(* CODESYS project PLCPID.project
   Title: PLCTEST
   Author: Peter
   Version: 0.0.0.21

Project tree, tasks and I/O mapping:
  MyController_1 : TM241CEC24T/U, Schneider Electric, order no. TM241CEC24T/U, version 4.0.6.18
    application Application
      libraries: HMISCU PTOPWM, 2.0.1.4 (Schneider Electric); SM3_Basic, 3.5.3.83 (3S - Smart Software Solutions GmbH)
      task MAST (cyclic, interval 2 ms, priority 15, watchdog 100 ms x 1) calls PIDController
      global variables GVL
      program PIDController [ST]
      function block Home [ST]
    DI : Digital Inputs, Schneider Electric, version 4.0.6.18
        settings: IOs Usage = 3
        input  Application.PIDController.sensor_r : BOOL  // IW0.I6
        input  Application.PIDController.sensor_l : BOOL  // IW0.I7
        input  ibDI_IB1 : BYTE  // IB1
        unmapped channels: IW0
    DQ : Digital Outputs, Schneider Electric, version 4.0.6.18
        output Application.PIDController.en_driver : BOOL  // QW0.Q7
        output Application.PIDController.fault_reset : BOOL  // QW0.Q8
        unmapped channels: QW0, QB1
    Counters : Counters, Schneider Electric, version 4.0.6.18
        settings: Instance name = 'encoder'; B input History = 'old=-1 new=1'; A input History = 'old=-1 new=0'; Temporary Instance name = 'encoder'
    Pulse_Generators : Pulse Generators, Schneider Electric, version 4.0.6.18
        settings: A output History = 'old=7 new=-1'
    Cartridge_1 : Cartridge, Schneider Electric, version 4.0.6.18
    IO_Bus : IO bus - TM3, Schneider Electric, version 4.0.6.18
      Module_1 : TM3SAF5R/G, Schneider Electric, order no. TM3SAF5R/G, version 1.0.1.12
          output Application.PIDController.en_safety : BOOL  // QB0.Enable
          unmapped channels: IW0, QB0
      Module_2 : TM3AQ4/G, Schneider Electric, order no. TM3AQ4/G, version 1.0.0.12
          settings: KPI Configuration.KPI Configuration[0] = 17; KPI Configuration.KPI Configuration[4] = 240; KPI Configuration.KPI Configuration[5] = 216; KPI Configuration.KPI Configuration[12] = 16; KPI Configuration.KPI Configuration[13] = 39
          output Application.PIDController.motor_value : INT  // QW0
          output qiModule_2_QW2 : INT  // QW2
          output qiModule_2_QW3 : INT  // QW3
          input  ibModule_2_IBStatusQW0 : BYTE  // IBStatusQW0
          input  ibModule_2_IBStatusQW1 : BYTE  // IBStatusQW1
          input  ibModule_2_IBStatusQW2 : BYTE  // IBStatusQW2
          input  ibModule_2_IBStatusQW3 : BYTE  // IBStatusQW3
          unmapped channels: QW1
    COM_Bus : COM bus, Schneider Electric, version 4.0.6.18
    Ethernet_1 : Ethernet Network, Schneider Electric, version 4.0.6.18
    Serial_Line_1 : Serial line, Schneider Electric, version 4.0.6.18
      Modbus_Manager : Modbus Manager, Schneider Electric, version 4.0.0.2
    Serial_Line_2 : Serial line, Schneider Electric, version 4.0.6.18
      Modbus_Manager1 : Modbus Manager, Schneider Electric, version 4.0.0.2
    CAN_1 : CANopen bus, Schneider Electric, version 4.0.6.18
      CANopen_Performance : CANopen Performance, Schneider Electric, order no. 1806, version 3.0.1.24
          settings: Heartbeat in Milliseconds = 100; ConfigVersion = 50659584
  FdtConnections : FDT Connections, Schneider Electric, version 1.0.0.2
    Modbus_Serial_Line_Manager : Modbus Serial Line Manager, Schneider Electric, version 2.2.5
      Lexium_32_C : Lexium 32 C Advanced Settings, Schneider Electric, version 1.14.02.00
  text list GlobalTextList
*)

// MyController_1/Application/GVL
VAR_GLOBAL
END_VAR

// MyController_1/Application/PIDController
PROGRAM PIDController
VAR
	error: REAL;
	o_analog: REAL;
	vel_pend: REAL;
	vel_mot: REAL;
	i_pos_mot: INT;
	i_pos_pend: INT;
	home: Home;
	sensor_l: BOOL;
	sensor_r: BOOL;
	i_ref_pos: INT;
	init: BOOL;
	last_error: REAL;
	ki: REAL;
	kp: REAL;
	kd: REAL;
	derivative: REAL;
	integral: REAL;
	fb_integral: INTEGRAL;
	integral_time: DWORD;
	motor_value: INT;
	home_timer: TON;
	en_safety: BOOL;
	en_driver: BOOL;
	fault_reset: BOOL;
	encoderValue: DINT;
	encoderValidate: BOOL;
	encoderError: EXPERTGetDiag;
END_VAR

IF NOT init THEN
	integral_time := 400;
	last_error := 0;
	
	home_timer.IN := FALSE;
	//Home time
	home_timer.PT := T#400MS;
	
	kp := 1;
	ki := 1;
	kd := 1;

	en_safety := TRUE;
	en_driver := TRUE;
	fault_reset := FALSE;	

	init := TRUE;
END_IF

Home(sensor_l := sensor_l, sensor_r := sensor_r, Fault := fault_reset, signal_out := motor_value);

(*
error := i_ref_pos - i_pos_pend;

fb_integral.IN := error;
fb_integral.TM := integral_time;
integral := fb_integral.OUT;

derivative := error - last_error;

o_analog := (kp * error) + (ki * integral) + (kd * derivative);

last_error := error;*)
encoderValue := encoder.CurrentValue;
encoder.Run;
encoderError.EXPERT_REF_IN := encoder.HSC_REF;
encoderError.Execute := TRUE;

encoderError();
encoder(EN_Enable:= TRUE, EN_Preset := TRUE, F_Preset := TRUE, F_Enable := TRUE);

END_PROGRAM

// MyController_1/Application/Home
FUNCTION_BLOCK Home
VAR_INPUT
	Execute: BOOL;
END_VAR
VAR_OUTPUT
	Done: BOOL;
END_VAR
VAR
	timer: TON;
END_VAR
VAR_IN_OUT
	signal_out: INT;
END_VAR
VAR_INPUT
	sensor_r: BOOL;
	sensor_l: BOOL;
END_VAR
VAR
	STATE: SINT := 0;
END_VAR
VAR_IN_OUT
	Fault: BOOL;
END_VAR
VAR
	timer_reset: TON;
	timer_reset_1: TON;
	timer_1: TON;
	temp_time: TIME;
	time_reset: REAL;
END_VAR

IF Execute THEN
CASE STATE OF
		0:
			signal_out := 3500;
			IF NOT sensor_r THEN
				signal_out := 0;
				timer_reset.IN := TRUE;
				
				IF timer_reset.Q THEN
					Fault := TRUE;
					STATE := 1;	
					timer_reset_1.IN := TRUE;
				END_IF
			END_IF
		1:
			timer_reset.IN := FALSE;
			IF timer_reset_1.Q THEN
				Fault := FALSE;
				timer.PT := T#100S;
				timer.IN := TRUE;
				signal_out := -3500;
				timer_reset_1.IN := FALSE;
			END_IF

			IF NOT sensor_l THEN
				time_reset := TIME_TO_REAL(timer.ET);
				timer_1.PT := (REAL_TO_TIME((TIME_TO_REAL(timer.ET)) / 2));
				signal_out := 0;
				timer_reset.IN := TRUE;
				
				IF timer_reset.Q THEN
					Fault := TRUE;
					timer_reset_1.IN := TRUE;
					STATE := 2;
				END_IF
			END_IF
		2:	
			timer_reset.IN := FALSE;
			
			IF timer_reset_1.Q THEN
				Fault := FALSE;
				timer_1.IN := TRUE;
				signal_out := 3500;
				timer_reset_1.IN := FALSE;
			END_IF
			
			IF timer_1.Q THEN
				signal_out := 0;
				Done := TRUE;
				Execute := FALSE;
			END_IF
END_CASE
timer();
timer_1();
timer_reset(PT := T#500MS);
timer_reset_1(PT := T#500MS);
END_IF

END_FUNCTION_BLOCK
